(* PLC project safeApp1, BrAutomation SafeDESIGNER  5.16.0.0 *)
(* stored: companyURL http://www.br-automation.com, creationDateTime Fri Mar 04 13:39:56 2022 *)

PROGRAM Main

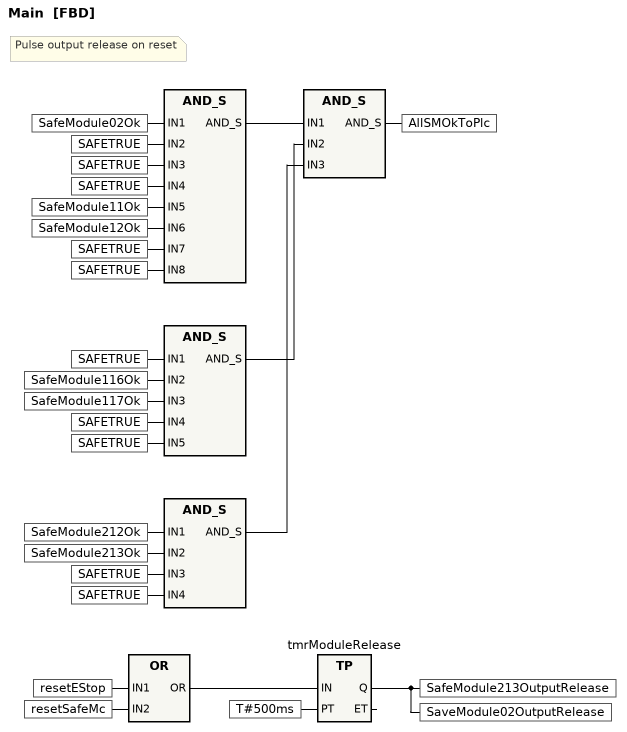
(* FBD diagram, written out as Structured Text *)
AllSMOkToPlc := AND_S(AND_S(SafeModule02Ok, SAFETRUE, SAFETRUE, SAFETRUE, SafeModule11Ok, SafeModule12Ok, SAFETRUE, SAFETRUE), AND_S(SAFETRUE, SafeModule116Ok, SafeModule117Ok, SAFETRUE, SAFETRUE), AND_S(SafeModule212Ok, SafeModule213Ok, SAFETRUE, SAFETRUE));
(* Pulse output release on reset *)
tmrModuleRelease(IN := resetEStop OR resetSafeMc, PT := T#500ms);
SafeModule213OutputRelease := tmrModuleRelease.Q;
SaveModule02OutputRelease := tmrModuleRelease.Q;
END_PROGRAM
